(* CODESYS project BagFeedSequence.Init_entry.xml

Project tree, tasks and I/O mapping:
*)

// Init_entry
ACTION Init_entry:
_attempts := 0;
END_ACTION
